FUNCTION_BLOCK Payload EXTENDS Serializable
VAR_INPUT
	timer : TON;
END_VAR
VAR_OUTPUT
END_VAR
VAR
	k : INT;	
END_VAR

timer();

END_FUNCTION_BLOCK

(* stored: Version 1.1.0.1, ProductVersion 3.1.4024.2
   POU Payload: Id {01decef4-4932-45b1-b8fd-b868843e0df2}, SpecialFunc None *)
